// TIA Portal V16 export
// export: Created 2023-03-29T11:04:49.9269314Z, ExportSetting WithDefaults, DisplayName Totally Integrated Automation Portal, DisplayVersion V16 Update 6, DisplayName TIA Portal Version Control Interface, DisplayVersion V16 Update 2, DisplayName TIA Portal Openness, DisplayVersion V16 Update 6, DisplayName STEP 7 Professional, DisplayVersion V16 Update 6, DisplayName STEP 7 Safety, DisplayVersion V16, DisplayName WinCC Advanced, DisplayVersion V16 Update 6
FUNCTION_BLOCK "Temp"   // FB22, LAD
{ S7_Optimized_Access := 'TRUE' }
VERSION : 0.1
// stored: AutoNumber true, IsIECCheckEnabled false, IsRetainMemResEnabled false, MemoryReserve 100, SetENOAutomatically false, UDAEnableTagReadback false
   VAR_INPUT
      Sub_PV_K1 : Real;   // Wspólczynnik pomniejszenia wyliczanego ciśnienia napotrzeby wyłączenia dodatowej pompy / Wspólczynnik pomniejszenia wyliczanego tlenu napotrzeby wyłączenia dodatowej dmuchawy
      InputWarning_H_PID { ExternalAccessible := 'False'; ExternalVisible := 'False'; ExternalWritable := 'False'} : Bool;   // Oszczerzenie górny limit
      InputWarning_L_PID { ExternalAccessible := 'False'; ExternalVisible := 'False'; ExternalWritable := 'False'} : Bool;   // Oczszczerzenie dolny limit
   END_VAR
   VAR_IN_OUT
      Set_K1 { ExternalWritable := 'False'} : Bool;   // Dostaw 1 dodatkową / Dostaw 1 dmuchawę dodatkową
   END_VAR
   VAR_TEMP
      Temp_SV_Int : Int;
   END_VAR
   VAR_TEMP   // added for the SCL form of the ladder/FBD networks
      _w1 : Bool;
      _w2 : Bool;
   END_VAR
BEGIN

REGION Network 1
   // OB 30 Network 14
END_REGION

REGION Network 2: Przekazanie wartości na wyjście analogowe "Out_Hz" -
   // Jeśli znacznik TmP_Set_SV (tymczasowe ustawienie Hz) wyłączony to na wyjście QW90 przekazywana jest wartość wyliczona z PID
   // Jeśli znacznik Tmp_Set_SV jest True to na wyjście przekazywana jest wartość tymczasowa 30Hz
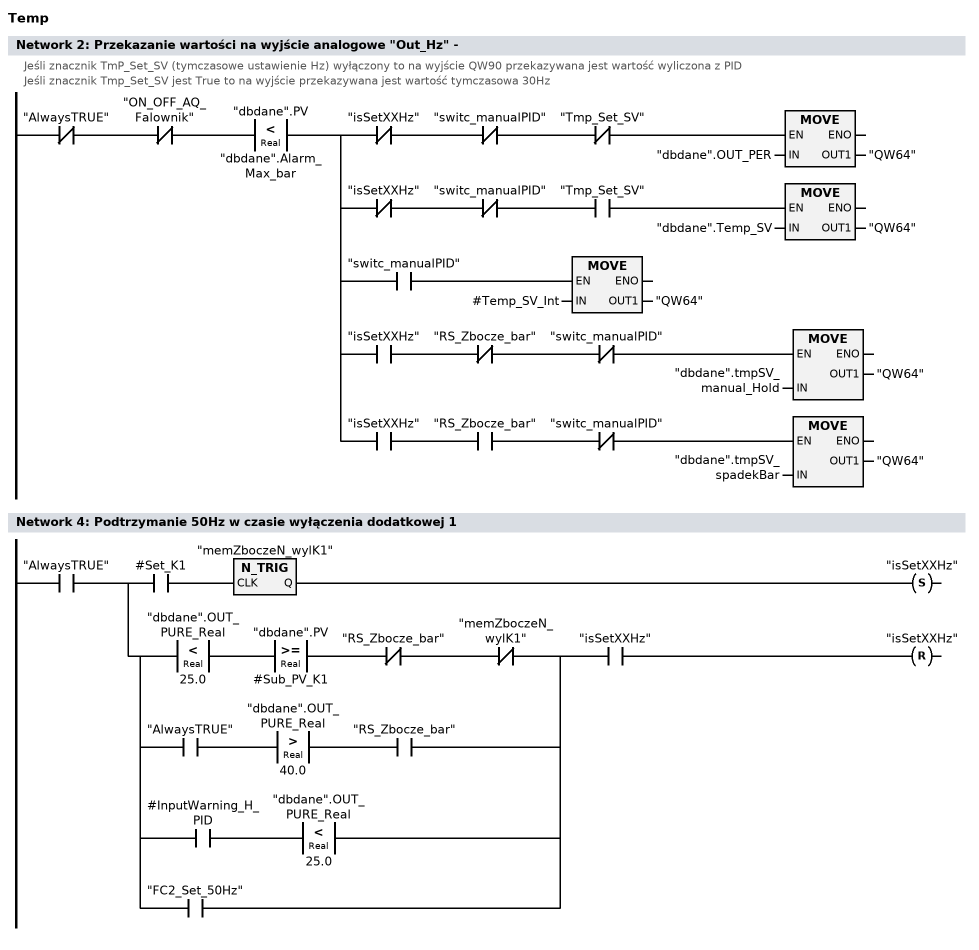
   RUNG wire#powerrail
      I_Contact( "AlwaysTRUE" )
      I_Contact( "ON_OFF_AQ_Falownik" )
      { S7_Templates := "SrcType := Real" } LT_Contact(in1 := "dbdane".PV, in2 := "dbdane".Alarm_Max_bar)
      wire#w1
      I_Contact( "isSetXXHz" )
      I_Contact( "switc_manualPID" )
      I_Contact( "Tmp_Set_SV" )
      { S7_GenerateENO := "TRUE" } Move(in := "dbdane".OUT_PER, out1 => "QW64")
   END_RUNG
   RUNG wire#w1
      I_Contact( "isSetXXHz" )
      I_Contact( "switc_manualPID" )
      Contact( "Tmp_Set_SV" )
      { S7_GenerateENO := "TRUE" } Move(in := "dbdane".Temp_SV, out1 => "QW64")
   END_RUNG
   RUNG wire#w1
      Contact( "switc_manualPID" )
      { S7_GenerateENO := "TRUE" } Move(in := #Temp_SV_Int, out1 => "QW64")
   END_RUNG
   RUNG wire#w1
      Contact( "isSetXXHz" )
      I_Contact( "RS_Zbocze_bar" )
      I_Contact( "switc_manualPID" )
      { S7_GenerateENO := "TRUE" } Move(in := "dbdane".tmpSV_manual_Hold, out1 => "QW64")
   END_RUNG
   RUNG wire#w1
      Contact( "isSetXXHz" )
      Contact( "RS_Zbocze_bar" )
      I_Contact( "switc_manualPID" )
      { S7_GenerateENO := "TRUE" } Move(in := "dbdane".tmpSV_spadekBar, out1 => "QW64")
   END_RUNG
   // the same network as SCL:
   #_w1 := NOT "AlwaysTRUE" AND NOT "ON_OFF_AQ_Falownik" AND ("dbdane".PV < "dbdane".Alarm_Max_bar);
   IF #_w1 AND NOT "isSetXXHz" AND NOT "switc_manualPID" AND NOT "Tmp_Set_SV" THEN
       "QW64" := "dbdane".OUT_PER;
   END_IF;
   IF #_w1 AND NOT "isSetXXHz" AND NOT "switc_manualPID" AND "Tmp_Set_SV" THEN
       "QW64" := "dbdane".Temp_SV;
   END_IF;
   IF #_w1 AND "switc_manualPID" THEN "QW64" := #Temp_SV_Int; END_IF;
   IF #_w1 AND "isSetXXHz" AND NOT "RS_Zbocze_bar" AND NOT "switc_manualPID" THEN
       "QW64" := "dbdane".tmpSV_manual_Hold;
   END_IF;
   IF #_w1 AND "isSetXXHz" AND "RS_Zbocze_bar" AND NOT "switc_manualPID" THEN
       "QW64" := "dbdane".tmpSV_spadekBar;
   END_IF;
END_REGION

REGION Network 3: FB1 Network 22
END_REGION

REGION Network 4: Podtrzymanie 50Hz w czasie wyłączenia dodatkowej 1
   RUNG wire#powerrail
      Contact( "AlwaysTRUE" )
      wire#w1
      Contact( #Set_K1 )
      N_Trig( "memZboczeN_wylK1" )
      S_Coil( "isSetXXHz" )
   END_RUNG
   RUNG wire#w1
      { S7_Templates := "SrcType := Real" } LT_Contact(in1 := "dbdane".OUT_PURE_Real, in2 := 25.0)
      { S7_Templates := "SrcType := Real" } GE_Contact(in1 := "dbdane".PV, in2 := #Sub_PV_K1)
      I_Contact( "RS_Zbocze_bar" )
      I_Contact( "memZboczeN_wylK1" )
      wire#w2
      Contact( "isSetXXHz" )
      R_Coil( "isSetXXHz" )
   END_RUNG
   RUNG wire#w1
      Contact( "AlwaysTRUE" )
      { S7_Templates := "SrcType := Real" } GT_Contact(in1 := "dbdane".OUT_PURE_Real, in2 := 40.0)
      Contact( "RS_Zbocze_bar" )
   END_RUNG wire#w2
   RUNG wire#w1
      Contact( #InputWarning_H_PID )
      { S7_Templates := "SrcType := Real" } LT_Contact(in1 := "dbdane".OUT_PURE_Real, in2 := 25.0)
   END_RUNG wire#w2
   RUNG wire#w1
      Contact( "FC2_Set_50Hz" )
   END_RUNG wire#w2
   // the same network as SCL:
   #_w1 := "AlwaysTRUE" AND #Set_K1;
   #_w2 := NOT #_w1 AND "memZboczeN_wylK1";   // falling edge
   "memZboczeN_wylK1" := #_w1;
   IF #_w2 THEN "isSetXXHz" := TRUE; END_IF;
   IF "AlwaysTRUE" AND ((("dbdane".OUT_PURE_Real < 25.0) AND ("dbdane".PV >= #Sub_PV_K1) AND NOT "RS_Zbocze_bar" AND NOT "memZboczeN_wylK1") OR ("AlwaysTRUE" AND ("dbdane".OUT_PURE_Real > 40.0) AND "RS_Zbocze_bar") OR (#InputWarning_H_PID AND ("dbdane".OUT_PURE_Real < 25.0)) OR "FC2_Set_50Hz") AND "isSetXXHz" THEN
       "isSetXXHz" := FALSE;
   END_IF;
END_REGION
END_FUNCTION_BLOCK
